// TIA Portal V16 export
// export: Created 2021-07-12T14:47:18.9564386Z, ExportSetting WithDefaults, DisplayName Totally Integrated Automation Portal, DisplayVersion V16, DisplayName TIA Portal Version Control Interface, DisplayVersion V16, DisplayName TIA Portal Openness, DisplayVersion V16, DisplayName STEP 7 Professional, DisplayVersion V16, DisplayName STEP 7 Safety, DisplayVersion V16, DisplayName WinCC Professional, DisplayVersion V16
TYPE "SimaHydTO_typeHMIConnectionAdvancedAxisControlStatus"
TITLE = SimaHydTO_typeHMIConnectionAdvancedAxisControlStatus
// HMI interface: Advanced axis control
// stored: IsFailsafeCompliant false
   STRUCT
      moveRelativeDone : Bool;   // MC_MoveRelative: Job is completed
      moveRelativeBusy : Bool;   // MC_MoveRelative: Job is running
      moveAbsoluteDone : Bool;   // MC_MoveAbsolute: Job is completed
      moveAbsoluteBusy : Bool;   // MC_MoveAbsolute: Job is running
      haltDone : Bool;   // MC_Halt: Job is running
      haltBusy : Bool;   // MC_Halt: Job is running
      commandAborted : Bool;   // The job was aborted by another job during execution (see also StatusID)
      error : Bool;   // An error occurred during execution of the job. The job is rejected. The cause of the error can be found in the "ErrorID" parameter.
      errorID : Word;   // ErrorID of motion control instruction (see also StatusID)
      statusID : Int;   // Additional specification of affected Motion control instruction of CommandAborted or Error: 0: No instruction / 1: MC_MoveRelative / 2: MC_MoveAbsolute / 3: MC_Halt
   END_STRUCT;
END_TYPE
